{attribute 'linkalways'} 
{attribute 'no_explicit_call' := 'This FB is a CLASS and must be accessed using methods or properties'}
{attribute 'enable_dynamic_creation'}
FUNCTION_BLOCK _INT EXTENDS NumericDatatypeBase
VAR
	localData : INT;
	activeData : REFERENCE TO INT REF= localData;
END_VAR

PROPERTY PUBLIC Address : PVOID
GET
Address := ADR(activeData);
END_GET
END_PROPERTY

METHOD PUBLIC ClearReference
VAR_INPUT
END_VAR
activeData REF= localData;
END_METHOD

METHOD PUBLIC Clone : I_Datatype
VAR
    pClone : POINTER TO _INT;
END_VAR
pClone := __NEW(_INT(InitialValue := Value));
Clone := pClone^;
END_METHOD

METHOD FB_init : BOOL
VAR_INPUT
	bInitRetains : BOOL; // if TRUE, the retain variables are initialized (warm start / cold start)
	bInCopyCode : BOOL;  // if TRUE, the instance afterwards gets moved into the copy code (online change)
	InitialValue : INT;
END_VAR
localData := InitialValue;
END_METHOD

PROPERTY PUBLIC IsFloat : BOOL
GET
IsFloat := FALSE;
END_GET
END_PROPERTY

PROPERTY PUBLIC IsSigned : BOOL
GET
IsSigned := TRUE;
END_GET
END_PROPERTY

METHOD PUBLIC MakeReferenceTo
VAR_INPUT
	ReferenceTarget : REFERENCE TO INT;
END_VAR
activeData REF= ReferenceTarget;
END_METHOD

PROPERTY PUBLIC MaxValue : INT
GET
MaxValue := DatatypeLimits.INT_MAX_VALUE;
END_GET
END_PROPERTY

PROPERTY PUBLIC MinValue : INT
GET
MinValue := DatatypeLimits.INT_MIN_VALUE;
END_GET
END_PROPERTY

METHOD PROTECTED SerializeMaxValue
VAR_INPUT
	Serializer : I_Serializer;
END_VAR
Serializer.AddInt(MaxValue);
END_METHOD

METHOD PROTECTED SerializeMinValue
VAR_INPUT
	Serializer : I_Serializer;
END_VAR
Serializer.AddInt(MinValue);
END_METHOD

METHOD PUBLIC SerializeWith
VAR_INPUT
	Serializer : I_Serializer;
END_VAR
Serializer.AddInt(activeData);
END_METHOD

PROPERTY PUBLIC Size : UDINT
GET
Size := SIZEOF(activeData);
END_GET
END_PROPERTY

METHOD TryDeserializeFrom : BOOL
VAR_INPUT
	Deserializer : I_Deserializer;
	Feedback : I_DeserializerFeedback;
END_VAR
TryDeserializeFrom := Deserializer.TryGetInt(activeData, Feedback);
END_METHOD

METHOD TryMakeReferenceTo : BOOL
VAR_INPUT
	Target : I_Datatype;
END_VAR
VAR
	pTargetData : POINTER TO INT;
END_VAR
IF NOT (Target.TypeName = TypeName) THEN
	RETURN;
END_IF

pTargetData := Target.Address;
activeData REF= pTargetData^;
TryMakeReferenceTo := TRUE;
END_METHOD

PROPERTY PUBLIC TypeName : T_MAXSTRING
GET
TypeName := 'INT';
END_GET
END_PROPERTY

PROPERTY PUBLIC Value : INT
GET
Value := activeData;
END_GET
SET
activeData := Value;
END_SET
END_PROPERTY

END_FUNCTION_BLOCK

(* stored: Version 1.1.0.1, ProductVersion 3.1.4024.12
   POU _INT: Id {c6e1a580-6260-05c7-3341-5c276fcad022}, SpecialFunc None
   Folder Constructor: Id {54966c0f-a60a-03f5-338f-4f59bf06139a}
   Folder Protected: Id {0ac54870-e0a8-06ee-32d2-4114a10ca736}
   Property Address: Id {c45218ca-5134-00c5-3b15-124c8940644c}
   Get Get: Id {aa814f67-3885-0961-3f7d-8dae8d278a39}
   Method ClearReference: Id {4325f9d2-5176-0f93-1ff0-c76b8ecdbc01}
   Method Clone: Id {1a9c0c20-14c9-0da4-17d0-fb20e097e2e8}
   Method FB_init: Id {26aa5e72-12cd-0881-2912-17aafaa6a3b6}
   Property IsFloat: Id {016f8bb9-68d4-0ec8-39c4-542f4b8bdb7b}
   Get Get: Id {3a480ef9-2ce4-014a-10d1-8753462c2b6a}
   Property IsSigned: Id {540c7438-4b0d-062f-3d40-158d23098cbf}
   Get Get: Id {0fed03fa-bd4e-04b4-2bf1-b760996a6d34}
   Method MakeReferenceTo: Id {0b18d376-cf26-00a1-295c-5c97bf30683a}
   Property MaxValue: Id {4fc83021-fbd1-0d32-3556-3c114106d000}
   Get Get: Id {d8285fd6-47ff-003f-02f2-1ab69f6785d6}
   Property MinValue: Id {dc757b64-1602-0ec5-2f49-2ce1f42686d4}
   Get Get: Id {b527509a-19b5-0c70-3ac9-4dd9c0bf7a62}
   Method SerializeMaxValue: Id {553c53b3-aa9b-0038-1498-e936cd1162d7}
   Method SerializeMinValue: Id {14d4ab00-c3d9-066e-35be-06b1ed5edf66}
   Method SerializeWith: Id {bf5fd625-b24d-03aa-1a7d-89fb7d78c094}
   Property Size: Id {68e7f418-94e3-0cbd-28ab-e770b35cbe67}
   Get Get: Id {38357b2e-8201-0997-3b5b-443ac1b2200f}
   Method TryDeserializeFrom: Id {e98a79ba-cb51-098f-27d6-0726e1838956}
   Method TryMakeReferenceTo: Id {4f59ba82-d14d-0dd0-29d4-b63510ddea7f}
   Property TypeName: Id {0df90c3f-b54b-044d-1c26-733911b9a0a8}
   Get Get: Id {37b7ff7c-35aa-0c25-185b-68ef14d3b7fe}
   Property Value: Id {a1480f1c-8fbd-09d1-0c8e-dc7a758ed390}
   Get Get: Id {55194669-b30a-0935-08e1-b1ab93916561}
   Set Set: Id {64ac6139-bae9-0c9b-31c1-3c422769556a} *)
